PROGRAM POU_OnFabrica
VAR
END_VAR

GVL_General.sBeltConveyor.bSortingCintaInicial := TRUE;
GVL_General.sBeltConveyor.bSortingCintaEntrada := TRUE;
GVL_General.sBeltConveyor.bSortingCintaDistribucion := TRUE;

GVL_General.sBeltConveyor.bCintaAzul2 := TRUE;
GVL_General.sBeltConveyor.bCintaVerde2 := TRUE;
GVL_General.sBeltConveyor.bCintaMetal2 := TRUE;

GVL_ProcesoPalet.sRollerConveyor.bRollerAlmacen1 := TRUE;
GVL_ProcesoPalet.sRollerConveyor.bRollerAlmacen2 := TRUE;
GVL_ProcesoPalet.sRollerConveyor.bCurvedRollerAlmacen := TRUE;

END_PROGRAM

(* stored: Version 1.1.0.1, ProductVersion 3.1.4024.12
   POU POU_OnFabrica: Id {0cb7f3fa-823d-4e17-9c09-7f7283f8c97d}, SpecialFunc None *)
